FUNCTION Map : REAL
VAR_INPUT
	fArg		: REAL; //x
	fInMin		: REAL;
	fInMax		: REAL;
	fOutMin		: REAL;
	fOutMax		: REAL;	
END_VAR
VAR
END_VAR

IF (fInMax - fInMin) <> 0 THEN
	Map := (((fArg - fInMin) * (fOutMax - fOutMin)) / (fInMax - fInMin)) + fOutMin;
END_IF

END_FUNCTION

(* stored: Version 1.1.0.1, ProductVersion 3.1.4024.6
   POU Map: Id {867a4e44-aff0-4348-8a24-0be96e3ada61}, SpecialFunc None *)
